// TIA Portal V20 export
DATA_BLOCK "E2MSimulation"   // DB23
{ DB_Accessible_From_OPC_UA := 'FALSE' }
// stored: DBAccessibleFromOPCUA false, DBAccessibleFromWebserver false, MemoryReserve 100
   VAR
      randomNumber : Real;   // Randomly generated number
   END_VAR
BEGIN
END_DATA_BLOCK
